{attribute 'GeneratedUsingTerminal: EL4008-0000-0018'}
{attribute addProperty BoxType "EL4008-0000-0018"}
{attribute addProperty Id "AO_Output_Channel_1AT %Q*AO_Output_Channel_BA7EBB7C2AO_Output_Channel_2AT %Q*AO_Output_Channel_BA7EBB7C2AO_Output_Channel_3AT %Q*AO_Output_Channel_BA7EBB7C2AO_Output_Channel_4AT %Q*AO_Output_Channel_BA7EBB7C2AO_Output_Channel_5AT %Q*AO_Output_Channel_BA7EBB7C2AO_Output_Channel_6AT %Q*AO_Output_Channel_BA7EBB7C2AO_Output_Channel_7AT %Q*AO_Output_Channel_BA7EBB7C2AO_Output_Channel_8AT %Q*AO_Output_Channel_BA7EBB7C2WcStateAT %I*WcState_0B2B16F91InfoDataAT %I*InfoData_94A18F5E2"}
{attribute addProperty CRC "2334429859"}
{attribute addProperty Size "19"}
TYPE EL4008_8B2492A3 EXTENDS EtcSlaveTerminalBase_947E5A46 :
STRUCT
	{attribute addProperty Name "AO_Output_Channel_1"}
	AO_Output_Channel_1 : AO_Output_Channel_BA7EBB7C;
	{attribute addProperty Name "AO_Output_Channel_2"}
	AO_Output_Channel_2 : AO_Output_Channel_BA7EBB7C;
	{attribute addProperty Name "AO_Output_Channel_3"}
	AO_Output_Channel_3 : AO_Output_Channel_BA7EBB7C;
	{attribute addProperty Name "AO_Output_Channel_4"}
	AO_Output_Channel_4 : AO_Output_Channel_BA7EBB7C;
	{attribute addProperty Name "AO_Output_Channel_5"}
	AO_Output_Channel_5 : AO_Output_Channel_BA7EBB7C;
	{attribute addProperty Name "AO_Output_Channel_6"}
	AO_Output_Channel_6 : AO_Output_Channel_BA7EBB7C;
	{attribute addProperty Name "AO_Output_Channel_7"}
	AO_Output_Channel_7 : AO_Output_Channel_BA7EBB7C;
	{attribute addProperty Name "AO_Output_Channel_8"}
	AO_Output_Channel_8 : AO_Output_Channel_BA7EBB7C;
	{attribute addProperty Name "WcState"}
	WcState : WcState_0B2B16F9;
	{attribute addProperty Name "InfoData"}
	InfoData : InfoData_94A18F5E;
END_STRUCT
END_TYPE

(* stored: Version 1.2.0.0, ProductVersion 3.1.4024.9
   DUT EL4008_8B2492A3: Id {c1895640-fe8b-4d3c-847e-89de1352523c} *)
